(* IEC 61131-3 sources: test/Class/SfcClass_InitStep, 1 file *)

(* ---- SfcClass_InitStep.st ---- *)
(*!
<Class
	Name               = "SfcClass_InitStep"
	Revision           = "0.0"
	RealtimeTask       = "false"
	CyclicTask         = "false"
	BackgroundTask     = "false"
	Sigmatek           = "false"
	OSInterface        = "false"
	HighPriority       = "false"
	Automatic          = "false"
	UpdateMode         = "Prescan"
	SharedCommandTable = "true"
	Objectsize         = "(284,120)">
	<Channels>
		<Client Name="Action0" Required="true" Internal="false"/>
	</Channels>
	<Network Name="SfcClass_InitStep">
		<!-- List of Components in this network -->
		<Components>
			<Object
				Name       = "_base"
				Class      = "Sfc_Step_Base"
				Position   = "(218,120)"
				Visualized = "true"
				Remotely   = "true">
				<Channels>
					<Server Name="Itf"/>
					<Server Name="T"/>
					<Server Name="X"/>
					<Client Name="CallTransition"/>
					<Client Name="LogonToInvoker"/>
				</Channels>
			</Object>
		</Components>
		<Comments>
		</Comments>
		<!-- List of Connections in this network -->
		<Connections>
			<Connection Source="this.Itf" Destination="_base.Itf" Vertices="(690,210),(518,210),"/>
			<Connection Source="this.X" Destination="_base.X" Vertices="(690,270),(518,270),"/>
			<Connection Source="this.T" Destination="_base.T" Vertices="(690,330),(518,330),"/>
			<Connection Source="_base.LogonToInvoker" Destination="this.LogonToInvoker" Vertices="(230,210),(38,210),"/>
			<Connection Source="_base.CallTransition" Destination="this.CallTransition" Vertices="(230,270),(38,270),"/>
		</Connections>
		<!-- Headerfiles -->
		<Options>
		</Options>
	</Network>
</Class>
*)
#pragma using Sfc_Step_Base

SfcClass_InitStep : CLASS
: Sfc_Step_Base
  //Servers:
  //Clients:
	Action0 	: CltChCmd_Sfc_Action_Base;
  //Variables:
  //Functions:
				//! <Function Name="OnActive" Hidden="true"/>
	FUNCTION VIRTUAL OnActive;
				//! <Function Name="OnInactive" Hidden="true"/>
	FUNCTION VIRTUAL OnInactive;
  //Tables:
	FUNCTION @STD
		VAR_OUTPUT
			ret_code	: CONFSTATES;
		END_VAR;
	FUNCTION GLOBAL TAB @CT_;
END_CLASS;

#pragma usingLtd Sfc_Action_Base

FUNCTION VIRTUAL SfcClass_InitStep::OnActive

	Action0.OnStepActive(ActionQualifier:=Sfc_Action_Base::N_QUALIFIER, TimerSetting:=0 ms);

	Action0.SetPriority(Priority:=0);

	Action0.UpdatePriorities();

END_FUNCTION
FUNCTION VIRTUAL SfcClass_InitStep::OnInactive

	Action0.OnStepInactive();

END_FUNCTION
